# EPICS SNL sequencer program: psmodbusEEIApp/src/unimagEEIControl.st
program unimagEEIControl

/*
 * EPICS State Notation Language program for UNIMAG interface
 * Handles automatic polarity switching and sequencing for EEI power supply
 *
 * Per the Modbus map, COMMAND WORD #1 bit 4 (CMD_START_RAMP) is documented
 * as "START_RAMP/TRIGGER" - a single, dual-purpose commit signal. Bits 5/6
 * (CMD_CURRENT_MODE_TRIG / CMD_CURRENT_MODE_SW) are a mutually-exclusive
 * mode selector (like polarity POS/NEG): "Software" mode applies register
 * writes immediately, "Triggered" mode requires CMD_START_RAMP to commit a
 * pending write - including a polarity switch, which otherwise has no
 * commit step of its own.
 *
 * The active mode is controlled live via "{P}:MODE_SW_ENABLE" (see
 * eei_ps_unimag.template - it also applies the mode to the hardware bits),
 * monitored here so it can be changed at runtime without restarting the IOC.
 *
 * Separately, per the EEI regulator firmware docs, quadrupole/normal-dipole
 * units switch polarity with physical contactors (CMD_POLARITY_POS/NEG_EXEC
 * + CMD_CONTACTORS_OPEN, confirmed via STAT_POLARITY_POS/NEG). This requires
 * ramping to zero and dropping to standby before the contactors can safely
 * move, then powering back on - see CHECK_STATE/RAMP_TO_ZERO/GO_STANDBY/
 * CHANGE_POLARITY/GO_POWERON below.
 *
 * The pulsed-dipole H-bridge regulator (e.g. DHPTB102) has no contactors and
 * is fully bipolar. There is no need to go to standby or sequence a
 * contactor - every setpoint update just writes the current reference and
 * pulses START_RAMP/TRIGGER (see SET_SIGNED_CURRENT below). This is
 * selected per-IOC by "{P}:CFG_POLARITY_VIA_SIGN" (set via the
 * POLARITY_VIA_SIGN db macro).
 *
 * Confirmed empirically (not just from documentation) that on this
 * topology, registers 40003-40004 (CURR_SET_RAW / CURRENT_SP_SIGN in
 * eei_ps.template) are actually a single 32-bit two's-complement current
 * reference at the wire level, not separate magnitude+sign fields as their
 * names/the Modbus map's column labels suggest: writing plain magnitude +
 * a 0/1 sign flag produces a large, wrong positive value for negative
 * setpoints (e.g. -1A firmware-reassembled as +66.536A, from
 * high_word=1, low_word=1000 -> 1*65536+1000). currentToRaw32() below
 * computes the correct 32-bit two's-complement split, written via the raw
 * CURR_SET_RAW32_LO/HI registers instead. This also matters for large
 * *positive* currents on this topology - e.g. above 65.535A - which
 * likewise don't fit in a single 16-bit word.
 *
 * The contactor units use the same register pair, but for the (unsigned)
 * magnitude only: verified on QUATB201 that low word 4464 + high word 1
 * drives 70A (1*65536+4464 mA; output voltage 105V), whereas writing the
 * magnitude as a plain 16-bit register (CURR_SET_RAW) silently truncates it
 * modulo 65.536A - a 100A request became 34.464A on every contactor unit.
 * The polarity of these units is still selected by the contactors, so only
 * the magnitude is written (WRITE_CURRENT_REF below).
 *
 * Every wait is bounded by "{P}:SET_TIMEOUT_S" and judged against the
 * tolerances "{P}:ZERO_TOLERANCE" (current considered zero before switching
 * polarity/standby) and "{P}:SET_TOLERANCE" (requested current considered
 * reached). Exact zero/setpoint are never reached on real hardware (sensor
 * noise, regulator dead-band), so a plain equality test would stall every
 * polarity change. A failed wait is reported through "{P}:ST_NOT_REACHED"
 * (a state - zero, standby, polarity or power-on - was not reached, MAJOR
 * STATE_RB) or "{P}:SP_NOT_REACHED" (the setpoint was not reached within
 * tolerance, MINOR STATE_RB). Both are cleared by the next setpoint or by
 * CMD_RESET.
 */

option +r;  /* Make reentrant */

/* C declarations */
%% #include <math.h>

/* Absolute difference, in Amps, between the readback and the requested
 * current. {P}:CURRENT_RB is the exact 32-bit readback, so this is a plain
 * difference: a unit that silently truncated the reference (e.g. a 16-bit
 * write above 65.535A) must show up as an error, not be masked. */
%% static double currentError(double rb, double sp)
%% {
%%     return fabs(rb - sp);
%% }

/* Splits a signed current in Amps into the 32-bit two's-complement raw
 * low/high words expected by the sign-bit/bipolar topology's combined
 * current-reference registers (see file header comment). */
%% static void currentToRaw32(double current_amps, int *lo, int *hi)
%% {
%%     int raw32 = (int)(current_amps * 1000.0 +
%%                        (current_amps >= 0 ? 0.5 : -0.5));
%%     *lo = raw32 & 0xFFFF;
%%     *hi = (raw32 >> 16) & 0xFFFF;
%% }

/* PV declarations */
double current_sp;
assign current_sp to "{P}:CURRENT_SP";
monitor current_sp;

double current_rb;
assign current_rb to "{P}:CURRENT_RB";
monitor current_rb;

int curr_set_raw32_lo;
assign curr_set_raw32_lo to "{P}:CURR_SET_RAW32_LO";

int curr_set_raw32_hi;
assign curr_set_raw32_hi to "{P}:CURR_SET_RAW32_HI";

int stat_polarity_pos;
assign stat_polarity_pos to "{P}:STAT_POLARITY_POS";
monitor stat_polarity_pos;

int stat_polarity_neg;
assign stat_polarity_neg to "{P}:STAT_POLARITY_NEG";
monitor stat_polarity_neg;

int stat_standby;
assign stat_standby to "{P}:STAT_STANDBY";
monitor stat_standby;

int stat_power_on;
assign stat_power_on to "{P}:STAT_POWER_ON";
monitor stat_power_on;

int cmd_standby;
assign cmd_standby to "{P}:CMD_STANDBY";

int cmd_power_on;
assign cmd_power_on to "{P}:CMD_POWER_ON";

int cmd_start_ramp;
assign cmd_start_ramp to "{P}:CMD_START_RAMP";

int mode_sw_enable;
assign mode_sw_enable to "{P}:MODE_SW_ENABLE";
monitor mode_sw_enable;

int polarity_via_sign;
assign polarity_via_sign to "{P}:CFG_POLARITY_VIA_SIGN";
monitor polarity_via_sign;

int cmd_contactors_open;
assign cmd_contactors_open to "{P}:CMD_CONTACTORS_OPEN";

int cmd_polarity_pos_exec;
assign cmd_polarity_pos_exec to "{P}:CMD_POLARITY_POS_EXEC";

int cmd_polarity_neg_exec;
assign cmd_polarity_neg_exec to "{P}:CMD_POLARITY_NEG_EXEC";

int cmd_reset;
assign cmd_reset to "{P}:CMD_RESET";
monitor cmd_reset;

double zero_tolerance;
assign zero_tolerance to "{P}:ZERO_TOLERANCE";
monitor zero_tolerance;

double set_tolerance;
assign set_tolerance to "{P}:SET_TOLERANCE";
monitor set_tolerance;

double set_timeout_s;
assign set_timeout_s to "{P}:SET_TIMEOUT_S";
monitor set_timeout_s;

int sp_not_reached;
assign sp_not_reached to "{P}:SP_NOT_REACHED";

int st_not_reached;
assign st_not_reached to "{P}:ST_NOT_REACHED";

/* Event flags */
evflag current_sp_ef;
sync current_sp current_sp_ef;

evflag cmd_reset_ef;
sync cmd_reset cmd_reset_ef;

/* State variables */
int requested_polarity;  /* 1=positive, 2=negative */
double requested_current;
double abs_current;
int polarity_change_needed;
int timeout_counter;

/* Constants */
#define TICK_S 0.5  /* wait states poll on this delay and count ticks */
#define TIMEOUT_TICKS ((int)(set_timeout_s / TICK_S))
#define POL_POSITIVE 1
#define POL_NEGATIVE 2

/* Writes a current magnitude/reference as the two 16-bit halves of the
 * 32-bit register pair 40003-40004 (both topologies, see file header). Both
 * words are written before the START_RAMP trigger commits them. */
#define WRITE_CURRENT_REF(amps) \
    currentToRaw32((amps), &curr_set_raw32_lo, &curr_set_raw32_hi); \
    pvPut(curr_set_raw32_lo); \
    pvPut(curr_set_raw32_hi)

/* Sequence step published to STATE_SM */
int sm_step;
assign sm_step to "{P}:STATE_SM_STEP";

/* STATE_SM values published in STATE_SM_STEP */
#define SM_READY     0
#define SM_GOTOSET   1
#define SM_GOTOSTATE 2
#define SM_GOZERO    3
#define SM_GOPOS     4
#define SM_GONEG     5

ss unimag_control {
    state IDLE {
        entry {
            sm_step = SM_READY;
            pvPut(sm_step);
        }

        when (efTestAndClear(current_sp_ef)) {
            /* New current setpoint received - a new attempt clears the
             * previous failure. */
            sp_not_reached = 0;
            pvPut(sp_not_reached);
            st_not_reached = 0;
            pvPut(st_not_reached);
            requested_current = current_sp;
            abs_current = fabs(requested_current);

            /* Determine requested polarity */
            if (requested_current >= 0) {
                requested_polarity = POL_POSITIVE;
            } else {
                requested_polarity = POL_NEGATIVE;
            }

            /* Check if polarity change is needed. Bipolar (polarity_via_sign)
             * units never need the contactor dance - every setpoint just
             * writes sign + magnitude and triggers (see CHECK_STATE). */
            if (polarity_via_sign) {
                polarity_change_needed = 0;
            } else {
                pvGet(stat_polarity_pos);
                pvGet(stat_polarity_neg);

                if ((requested_polarity == POL_POSITIVE && !stat_polarity_pos) ||
                    (requested_polarity == POL_NEGATIVE && !stat_polarity_neg)) {
                    polarity_change_needed = 1;
                    timeout_counter = 0;
                } else {
                    polarity_change_needed = 0;
                }
            }
        } state CHECK_STATE

        when (efTestAndClear(cmd_reset_ef)) {
            /* Reset command cancels all operations and clears failures */
            polarity_change_needed = 0;
            timeout_counter = 0;
            sp_not_reached = 0;
            pvPut(sp_not_reached);
            st_not_reached = 0;
            pvPut(st_not_reached);
        } state IDLE
    }

    state CHECK_STATE {
        entry {
            /* Get current status */
            pvGet(stat_power_on);
            pvGet(current_rb);
        }

        when (polarity_via_sign) {
            /* Bipolar H-bridge unit: no contactors/standby to sequence -
             * just write sign + magnitude and trigger. */
        } state SET_SIGNED_CURRENT

        when (!polarity_change_needed) {
            /* No polarity change needed, just set current directly */
        } state SET_CURRENT_DIRECT

        when (polarity_change_needed && stat_power_on && fabs(current_rb) > zero_tolerance) {
            /* Need to ramp to zero first */
        } state RAMP_TO_ZERO

        when (polarity_change_needed && stat_power_on && fabs(current_rb) <= zero_tolerance) {
            /* Zero within tolerance, can go directly to standby */
        } state GO_STANDBY

        when (polarity_change_needed && !stat_power_on) {
            /* Already in standby or off, can change polarity */
        } state CHANGE_POLARITY
    }

    state RAMP_TO_ZERO {
        entry {
            sm_step = SM_GOZERO;
            pvPut(sm_step);
            /* Set current to zero and start ramp */
            WRITE_CURRENT_REF(0.0);
            cmd_start_ramp = 1;
            pvPut(cmd_start_ramp);
            timeout_counter = 0;
        }

        when (fabs(current_rb) <= zero_tolerance) {
            /* Current reached zero (within tolerance) */
        } state GO_STANDBY

        when (timeout_counter >= TIMEOUT_TICKS) {
            /* Timeout - cancel operation */
            polarity_change_needed = 0;
            st_not_reached = 1;
            pvPut(st_not_reached);
            printf("unimagControl: Zero not reached (current=%.3fA, tolerance=%.3fA)\n",
                   current_rb, zero_tolerance);
        } state IDLE

        when (efTestAndClear(cmd_reset_ef)) {
            polarity_change_needed = 0;
        } state IDLE

        when (delay(TICK_S)) {
            /* Keep checking */
            timeout_counter++;
        } state RAMP_TO_ZERO
    }

    state GO_STANDBY {
        entry {
            sm_step = SM_GOTOSTATE;
            pvPut(sm_step);
            cmd_standby = 1;
            pvPut(cmd_standby);
            timeout_counter = 0;
        }

        when (delay(0.5)) {
        } state WAIT_STANDBY
    }

    state WAIT_STANDBY {
        when (stat_standby) {
            /* Standby confirmed */
        } state CHANGE_POLARITY

        when (timeout_counter >= TIMEOUT_TICKS) {
            /* Timeout - cancel operation */
            polarity_change_needed = 0;
            st_not_reached = 1;
            pvPut(st_not_reached);
            printf("unimagControl: Standby not reached\n");
        } state IDLE

        when (efTestAndClear(cmd_reset_ef)) {
            polarity_change_needed = 0;
        } state IDLE

        when (delay(TICK_S)) {
            /* Keep checking */
            timeout_counter++;
        } state WAIT_STANDBY
    }

    state CHANGE_POLARITY {
        entry {
            sm_step = (requested_polarity == POL_POSITIVE) ? SM_GOPOS : SM_GONEG;
            pvPut(sm_step);
            /* Contactor-based units only (bipolar/polarity_via_sign units
             * are dispatched straight to SET_SIGNED_CURRENT and never reach
             * this state) - open contactors first. */
            cmd_contactors_open = 1;
            pvPut(cmd_contactors_open);
            timeout_counter = 0;
        }

        when (delay(1.0)) {
            /* Change polarity after delay. This register is a mutually-
             * exclusive selector (OPEN/POS/NEG), so a plain write of 1 or 2
             * replaces the whole register, clearing OPEN and the other
             * polarity bit in one atomic Modbus write. */
            if (requested_polarity == POL_POSITIVE) {
                cmd_polarity_pos_exec = 1;
                pvPut(cmd_polarity_pos_exec);
            } else {
                cmd_polarity_neg_exec = 2;
                pvPut(cmd_polarity_neg_exec);
            }
            /* In Triggered mode, the polarity write above has no commit of
             * its own - pulse the START_RAMP/TRIGGER bit to apply it. */
            if (!mode_sw_enable) {
                cmd_start_ramp = 1;
                pvPut(cmd_start_ramp);
            }
        } state WAIT_POLARITY_DELAY
    }

    state WAIT_POLARITY_DELAY {
        entry {
            timeout_counter = 0;
        }

        when (delay(2.0)) {
        } state WAIT_POLARITY
    }

    state WAIT_POLARITY {
        entry {
            pvGet(stat_polarity_pos);
            pvGet(stat_polarity_neg);
        }

        when ((requested_polarity == POL_POSITIVE && stat_polarity_pos) ||
              (requested_polarity == POL_NEGATIVE && stat_polarity_neg)) {
            /* Polarity confirmed */
            polarity_change_needed = 0;
        } state GO_POWERON

        when (timeout_counter >= TIMEOUT_TICKS) {
            /* Timeout - cancel operation */
            polarity_change_needed = 0;
            st_not_reached = 1;
            pvPut(st_not_reached);
            printf("unimagControl: Polarity change not reached\n");
        } state IDLE

        when (efTestAndClear(cmd_reset_ef)) {
            polarity_change_needed = 0;
        } state IDLE

        when (delay(TICK_S)) {
            /* Keep checking */
            timeout_counter++;
            pvGet(stat_polarity_pos);
            pvGet(stat_polarity_neg);
        } state WAIT_POLARITY
    }

    state GO_POWERON {
        entry {
            sm_step = SM_GOTOSTATE;
            pvPut(sm_step);
            cmd_power_on = 1;
            pvPut(cmd_power_on);
            timeout_counter = 0;
        }

        when (delay(0.5)) {
        } state WAIT_POWERON
    }

    state WAIT_POWERON {
        when (stat_power_on) {
            /* Power on confirmed */
        } state SET_CURRENT

        when (timeout_counter >= TIMEOUT_TICKS) {
            /* Timeout - cancel operation */
            st_not_reached = 1;
            pvPut(st_not_reached);
            printf("unimagControl: Power on not reached\n");
        } state IDLE

        when (efTestAndClear(cmd_reset_ef)) {
        } state IDLE

        when (delay(TICK_S)) {
            /* Keep checking */
            timeout_counter++;
        } state WAIT_POWERON
    }

    state SET_CURRENT {
        entry {
            sm_step = SM_GOTOSET;
            pvPut(sm_step);
            /* Set the absolute current value */
            WRITE_CURRENT_REF(abs_current);
        }

        when (delay(0.5)) {
        } state START_RAMP
    }

    state START_RAMP {
        entry {
            cmd_start_ramp = 1;
            pvPut(cmd_start_ramp);
        }

        when (delay(0.2)) {
        } state VERIFY_SET
    }

    state SET_CURRENT_DIRECT {
        entry {
            sm_step = SM_GOTOSET;
            pvPut(sm_step);
            /* No polarity change needed, check if we need to power on */
            pvGet(stat_power_on);
            timeout_counter = 0;
        }

        when (!stat_power_on) {
            /* Need to power on first */
            cmd_power_on = 1;
            pvPut(cmd_power_on);
        } state WAIT_POWERON_DIRECT

        when (stat_power_on) {
            /* Already powered on */
            WRITE_CURRENT_REF(abs_current);
        } state RAMP_DIRECT
    }

    state WAIT_POWERON_DIRECT {
        entry {
            sm_step = SM_GOTOSTATE;
            pvPut(sm_step);
        }

        when (stat_power_on) {
            WRITE_CURRENT_REF(abs_current);
        } state RAMP_DIRECT

        when (timeout_counter >= TIMEOUT_TICKS) {
            /* Timeout - don't get stuck here forever, or every future
             * setpoint would silently be ignored (IDLE never revisited). */
            st_not_reached = 1;
            pvPut(st_not_reached);
            printf("unimagControl: Power on not reached (direct)\n");
        } state IDLE

        when (efTestAndClear(cmd_reset_ef)) {
        } state IDLE

        when (delay(TICK_S)) {
            /* Keep checking */
            timeout_counter++;
        } state WAIT_POWERON_DIRECT
    }

    state RAMP_DIRECT {
        entry {
            sm_step = SM_GOTOSET;
            pvPut(sm_step);
        }

        when (delay(0.5)) {
            cmd_start_ramp = 1;
            pvPut(cmd_start_ramp);
        } state IDLE_DIRECT
    }

    state IDLE_DIRECT {
        when (delay(0.2)) {
        } state VERIFY_SET
    }

    state SET_SIGNED_CURRENT {
        entry {
            sm_step = SM_GOTOSET;
            pvPut(sm_step);
            /* Bipolar H-bridge unit: reverse current electronically via the
             * 32-bit two's-complement current reference - no contactors, no
             * standby, no ramp-to-zero. Write the complete signed reference
             * up front (see currentToRaw32, file header); only power-on is
             * state-dependent from here. */
            currentToRaw32(requested_current, &curr_set_raw32_lo, &curr_set_raw32_hi);
            pvPut(curr_set_raw32_lo);
            pvPut(curr_set_raw32_hi);
            pvGet(stat_power_on);
            timeout_counter = 0;
        }

        when (!stat_power_on) {
            /* Need to power on first */
            cmd_power_on = 1;
            pvPut(cmd_power_on);
        } state WAIT_POWERON_SIGNED

        when (stat_power_on) {
            /* Already powered on, reference already written above */
        } state RAMP_SIGNED
    }

    state WAIT_POWERON_SIGNED {
        entry {
            sm_step = SM_GOTOSTATE;
            pvPut(sm_step);
        }

        when (stat_power_on) {
            /* Reference already written in SET_SIGNED_CURRENT's entry */
        } state RAMP_SIGNED

        when (timeout_counter >= TIMEOUT_TICKS) {
            /* Timeout - don't get stuck here forever, or every future
             * setpoint would silently be ignored (IDLE never revisited). */
            st_not_reached = 1;
            pvPut(st_not_reached);
            printf("unimagControl: Power on not reached (signed)\n");
        } state IDLE

        when (efTestAndClear(cmd_reset_ef)) {
        } state IDLE

        when (delay(TICK_S)) {
            /* Keep checking */
            timeout_counter++;
        } state WAIT_POWERON_SIGNED
    }

    state RAMP_SIGNED {
        entry {
            sm_step = SM_GOTOSET;
            pvPut(sm_step);
        }

        when (delay(0.5)) {
            cmd_start_ramp = 1;
            pvPut(cmd_start_ramp);
        } state IDLE_SIGNED
    }

    state IDLE_SIGNED {
        when (delay(0.2)) {
        } state VERIFY_SET
    }

    /* Waits for the readback to get within SET_TOLERANCE of the requested
     * current. A SET_TOLERANCE of 0 disables the check. A new setpoint or a
     * reset abandons the wait (IDLE then consumes the pending event). */
    state VERIFY_SET {
        entry {
            sm_step = SM_GOTOSET;
            pvPut(sm_step);
            timeout_counter = 0;
        }

        when (set_tolerance <= 0) {
        } state IDLE

        when (efTest(current_sp_ef) || efTest(cmd_reset_ef)) {
        } state IDLE

        when (currentError(current_rb, requested_current) <= set_tolerance) {
            /* Setpoint reached (within tolerance) */
        } state IDLE

        when (timeout_counter >= TIMEOUT_TICKS) {
            sp_not_reached = 1;
            pvPut(sp_not_reached);
            printf("unimagControl: Setpoint not reached (requested=%.3fA, readback=%.3fA, tolerance=%.3fA)\n",
                   requested_current, current_rb, set_tolerance);
        } state IDLE

        when (delay(TICK_S)) {
            /* Keep checking */
            timeout_counter++;
        } state VERIFY_SET
    }
}
